PROGRAM PLC_PowerRF
VAR_INPUT
	nSocketType:UINT:=0;// socket 类型; 0 表示 server; 1 表示 client;
	sTerminalName:STRING;// 通讯对方名称 自定义
	sHost:STRING(20):='127.0.0.1';// 通讯IP地址; server时表示本地host; client时表示远程host
	nPort:UDINT:=8900;// 通讯端口号;
	bEnable:BOOL:=TRUE;// 通讯启用\禁用连接
	sSendSuffix:STRING:='';//此处可统一添加发送后缀字符 $R$N
	nQueueInterval:UDINT:=50;// 发送队列时间间隔 单位ms
	logHandleArray:ARRAY [1..5] OF POINTER TO printLogModule_EX;// log 操作 handle 数组
	logHandleArrayLength:UINT:=0;// log 操作 handle 数组长度, 不超过5
	readStateFlag:BOOL;
	ClearCom:BOOL;
	receiveFlag:BOOL;
END_VAR
VAR_OUTPUT
	bSendCondition	:BOOL;//可发送条件
	bSocketConnected:BOOL;//连接状态
END_VAR
VAR CONSTANT
	cNumBegin		:DINT:=1;
	cNumEnd			:DINT:=100;
END_VAR
VAR
	sendDataArray	:ARRAY [cNumBegin..cNumEnd] OF STRING(255);
	length			:DINT:=0;
	endPoint		:DINT:=cNumBegin;
	popupSendData	:STRING(255);
	//popup
	popupStep		:UINT:=0;
	popupTON1		:TON;
	popupTON2		:TON;
	iPopup			:DINT:=0;
	_PopupLength	:DINT:=0;
END_VAR
VAR
	tcpipClient					:tcpipClientModule_EX;
	tcpipServer					:tcpipServerModule_EX;////定义服务器对象
	
	tcpipSendDataBuff_Server	:STRING(255);//发送数据 Buff server
	tcpipSendDataBuff_Client	:STRING(255);//发送数据 Buff client
	
	tcpipSendDataClear			:STRING(255);//发送数据 清空
	tcpipSendData				:STRING(255);//发送数据
	
	tcpipRecDataBuff_Server		:STRING(255);//已接收数据 Buff server
	tcpipRecDataBuff_Client		:STRING(255);//已接收数据 Buff client
	
	tcpipRecDataClear			:STRING(255);//已接收数据 清空
	tcpipRecData				:STRING(255);//已接收数据
	
	tcpConnectR_Trig			:R_Trig;//初始连接上升沿
	tcpConnectF_Trig			:F_Trig;//初始连接下降沿
	registerStep				:UDINT;//ALC注册控制步
	registerTON					:TON;//ALC注册延时
	
	logHandleArray_index		:UINT:=1;
END_VAR
VAR
	bTrig_Start:BOOL;
	rTrig_Start:R_TRIG;
	tTrig_Start:TON;
	
	bTrig_Stop:BOOL;
	rTrig_Stop:R_TRIG;
	tTrig_Stop:TON;
	
	bTrig_Reset:BOOL;
	rTrig_Reset:R_TRIG;
	tTrig_Reset:TON;
	
	
	bTrig_Init:BOOL;
	rTrig_Init:R_TRIG;
	
	bTrig_All_Home:BOOL;
	rTrig_All_Home:R_TRIG;
	
	bTrig_Z_Safe:BOOL;
	rTrig_Z_Safe:R_TRIG;
	
	bTrig_P_Pos_:BOOL;
	rTrig_P_Pos_:R_TRIG;
	nTrig_P_Pos_TrayNum:UINT:=1;
	nTrig_P_Pos_RowNum:UINT:=1;
	
	bTrig_Move_P_:BOOL;
	rTrig_Move_P_:R_TRIG;
	nTrig_Move_P_TrayNum:UINT:=1;
	nTrig_Move_P_RowNum:UINT:=1;
	nTrig_Move_P_PosNum:UINT:=1;
	findposstart	:INT;
	findposend		:INT;
	find_pos		:INT;
	recStrTemp		:STRING(255);
END_VAR


CASE nSocketType OF
0://TCPIP server
	tcpipServer(
		sSrvNetId:= , 
		sLocalHost:=sHost , 
		nLocalPort:=nPort , 
		bStartConnect:=bEnable , 
		tcpipSDataLen:=TO_UDINT(LEN(tcpipSendDataBuff_Server)) , 
		tcpipSData:=ADR(tcpipSendDataBuff_Server) , 
		bSend:= , 
		tcpipRecDataLen:=SIZEOF(tcpipRecDataBuff_Server) , 
		tcpipRecData:=ADR(tcpipRecDataBuff_Server) , 
		bAccepted=> , 
		bSendBusy=> , 
		bRecData=> );
	bSendCondition:=tcpipServer.bAccepted AND NOT tcpipServer.bSendBusy;
	//TCPIP连接
	bSocketConnected:=tcpipServer.bAccepted;
	IF NOT tcpipServer.bAccepted THEN
		length:=0;
		endPoint:=cNumBegin;
	END_IF
	tcpConnectR_Trig(CLK:=tcpipServer.bAccepted);
	tcpConnectF_Trig(CLK:=tcpipServer.bAccepted);

1://TCPIP client
	tcpipClient(
		sSrvNetId:= , 
		sRemoteHost:=sHost , 
		nRemotePort:=nPort , 
		bStartConnect:=bEnable , 
		tcpipSDataLen:=TO_UDINT(LEN(tcpipSendDataBuff_Client)) , 
		tcpipSData:=ADR(tcpipSendDataBuff_Client) , 
		bSend:= , 
		tcpipRecDataLen:=SIZEOF(tcpipRecDataBuff_Client) , 
		tcpipRecData:=ADR(tcpipRecDataBuff_Client) , 
		bConnected=> , 
		bSendBusy=> , 
		bRecData=> );
	bSendCondition:=tcpipClient.bConnected AND NOT tcpipClient.bSendBusy;
	//TCPIP连接
	bSocketConnected:=tcpipClient.bConnected;
	IF NOT tcpipClient.bConnected THEN
		length:=0;
		endPoint:=cNumBegin;
	END_IF
	tcpConnectR_Trig(CLK:=tcpipClient.bConnected);
	tcpConnectF_Trig(CLK:=tcpipClient.bConnected);
END_CASE
IF ClearCom THEN
	length:=0;
	endPoint:=cNumBegin;
	ClearCom:=FALSE;
END_IF
IF tcpConnectR_Trig.Q THEN
	FOR logHandleArray_index:=1 TO logHandleArrayLength DO
		logHandleArray[logHandleArray_index]^.append(CONCAT(sTerminalName, ' has been connected'));
	END_FOR
	registerStep:=10;
END_IF
IF tcpConnectF_Trig.Q THEN
	FOR logHandleArray_index:=1 TO logHandleArrayLength DO
		logHandleArray[logHandleArray_index]^.append(CONCAT(sTerminalName, ' has been disconnected'));
	END_FOR
	registerStep:=0;
END_IF
//数据接收处理
CASE nSocketType OF
0://TCPIP server
	IF tcpipServer.bRecData THEN
		tcpipRecData:=tcpipRecDataBuff_Server;//buff转存
		tcpipRecDataBuff_Server:=tcpipRecDataClear;//转存之后清空buff
		dataProcessing();
	END_IF
1://TCPIP client
	IF tcpipClient.bRecData THEN
		tcpipRecData:=tcpipRecDataBuff_Client;//buff转存
		tcpipRecDataBuff_Client:=tcpipRecDataClear;//转存之后清空buff
		dataProcessing();
	END_IF
END_CASE


popup();

CASE registerStep OF
0:
	//Ready
END_CASE

METHOD appendSend : BOOL
VAR_INPUT
	str			:STRING(255);
END_VAR
VAR
	suffix					:STRING;
	strTemp_appendSend		:STRING(255);
END_VAR

IF endPoint>(cNumEnd-1) THEN
	RETURN;
END_IF
suffix:=sSendSuffix;//此处可统一添加发送后缀字符 $R$N

strTemp_appendSend:=CONCAT(str,suffix);
sendDataArray[endPoint]:=strTemp_appendSend;

endPoint:=endPoint+1;
length:=endPoint-cNumBegin;
END_METHOD

METHOD dataProcessing : BOOL
VAR_INPUT
END_VAR
VAR
	strTemp:STRING;
END_VAR
FOR logHandleArray_index:=1 TO logHandleArrayLength DO
	CASE nSocketType OF
	0://TCPIP server
//		logHandleArray[logHandleArray_index]^.append(CONCAT(CONCAT(CONCAT('Recevie From ', sTerminalName), ' -- '),tcpipRecData));
	1://TCPIP client
//		logHandleArray[logHandleArray_index]^.append(CONCAT(CONCAT(CONCAT('Recevie From ', sTerminalName), ' -- '),tcpipRecData));
	END_CASE
END_FOR
receiveFlag:=TRUE;
findposend:=0;
find_pos:=0;
IF MID(tcpipRecData,1,32)='$R' AND MID(tcpipRecData,1,33)='$R'  THEN
	gICP.PowerRF.controlMode:=STRING_TO_INT(MID(tcpipRecData,1,1));
	gICP.PowerRF.outputMode:=STRING_TO_INT(MID(tcpipRecData,1,2));
	gICP.PowerRF.outputState:=STRING_TO_INT(MID(tcpipRecData,1,3));
	strTemp:='';
	strTemp:=CONCAT(strTemp,(MID(tcpipRecData,2,6)));
	gICP.PowerRF.alarmState:=STRING_TO_INT(strTemp);
	strTemp:='';
	strTemp:=CONCAT(strTemp,(MID(tcpipRecData,5,9)));
	gICP.PowerRF.setpowerRead:=STRING_TO_UDINT(strTemp);
	strTemp:='';
	strTemp:=CONCAT(strTemp,(MID(tcpipRecData,5,15)));
	gICP.PowerRF.forwardpower:=STRING_TO_UDINT(strTemp);
	strTemp:='';
	strTemp:=CONCAT(strTemp,(MID(tcpipRecData,5,21)));
	gICP.PowerRF.reflectedpower:=STRING_TO_UDINT(strTemp);
	strTemp:='';
	strTemp:=CONCAT(strTemp,(MID(tcpipRecData,5,27)));
	gICP.PowerRF.maxpower:=STRING_TO_UDINT(strTemp);
	readStateFlag:=TRUE;
END_IF
END_METHOD

METHOD PRIVATE popup : BOOL
VAR_INPUT
END_VAR
CASE popupStep OF
0:
	IF length>0 AND bSendCondition THEN
		_PopupLength:=length;
		popupSendData:=sendDataArray[cNumBegin];
		FOR iPopup:=cNumBegin TO (_PopupLength-1) DO
			sendDataArray[iPopup]:=sendDataArray[iPopup+1];
		END_FOR
		endPoint:=endPoint-1;
		length:=endPoint-cNumBegin;
		sendData(popupSendData);//此处是调用信息发送
		popupStep:=10;
	END_IF
10:
	popupTON2(IN:=NOT popupTON2.Q, PT:=T#2S);
	IF NOT bSendCondition OR popupTON2.Q THEN
		popupTON2(IN:=FALSE);
		popupStep:=11;
	END_IF
11:
	IF bSendCondition THEN
		popupStep:=12;
	END_IF
	popupTON1(IN:=FALSE);
12:
	//popupTON1(IN:=NOT popupTON1.Q,PT:=T#10MS);
	popupTON1(IN:=NOT popupTON1.Q,PT:=TO_TIME(nQueueInterval));
	IF popupTON1.Q THEN
		popupStep:=0;
	END_IF
END_CASE
END_METHOD

METHOD ReadState : BOOL
VAR_INPUT
END_VAR
VAR
END_VAR
appendSend('Q$R');
END_METHOD

METHOD PRIVATE sendData : BOOL
VAR_INPUT
	dataStruct	:STRING(255);
END_VAR
IF bSendCondition AND bEnable THEN
	tcpipSendData:=dataStruct;
	
	CASE nSocketType OF
	0://TCPIP server
		tcpipSendDataBuff_Server:=tcpipSendData;
		tcpipSendData:=tcpipSendDataClear;	
		tcpipServer.bSend:=TRUE;
	1://TCPIP client
		tcpipSendDataBuff_Client:=tcpipSendData;
		tcpipSendData:=tcpipSendDataClear;	
		tcpipClient.bSend:=TRUE;
	END_CASE
	
	FOR logHandleArray_index:=1 TO logHandleArrayLength DO
		CASE nSocketType OF
		0://TCPIP server
//			logHandleArray[logHandleArray_index]^.append(CONCAT(CONCAT(CONCAT('Send To ', sTerminalName), ' -- '),tcpipSendDataBuff_Server));
		1://TCPIP client
//			logHandleArray[logHandleArray_index]^.append(CONCAT(CONCAT(CONCAT('Send To ', sTerminalName), ' -- '),tcpipSendDataBuff_Client));
		END_CASE
	END_FOR
END_IF
END_METHOD

METHOD WriteMaxPower : BOOL
VAR_INPUT
	maxpowerpoint:UDINT;
END_VAR
VAR
	str:STRING;
	_bit:UDINT;
	_ten:UDINT;
	_hundred:UDINT;
	_thousand:UDINT;
END_VAR
str:='';
_thousand:=maxpowerpoint/1000;
str:=CONCAT(str,UDINT_TO_STRING(maxpowerpoint));
//_hundred:=maxpowerpoint/100 MOD 10;
//str:=CONCAT(str,UDINT_TO_STRING(_hundred));
//_ten:=maxpowerpoint/10 MOD 10;
//str:=CONCAT(str,UDINT_TO_STRING(_ten));
//_bit:=maxpowerpoint MOD 10;
//str:=CONCAT(str,UDINT_TO_STRING(_bit));
str:=CONCAT(str,' M$R');
appendSend(str);
END_METHOD

METHOD WritePower : BOOL
VAR_INPUT
	powerpoint:UDINT;
END_VAR
VAR
	str:STRING;
	_bit:UDINT;
	_ten:UDINT;
	_hundred:UDINT;
	_thousand:UDINT;
END_VAR
str:='';
//_thousand:=powerpoint/1000;
str:=CONCAT(str,UDINT_TO_STRING(powerpoint));
//_hundred:=powerpoint/100 MOD 10;
//str:=CONCAT(str,UDINT_TO_STRING(_hundred));
//_ten:=powerpoint/10 MOD 10;
//str:=CONCAT(str,UDINT_TO_STRING(_ten));
//_bit:=powerpoint MOD 10;
//str:=CONCAT(str,UDINT_TO_STRING(_bit));
str:=CONCAT(str,' W$R');
appendSend(str);
END_METHOD

METHOD WriteReset : BOOL
VAR_INPUT
		

END_VAR
appendSend('RESET$R');
END_METHOD

METHOD WriteRS232Mode : BOOL
VAR_INPUT
		

END_VAR
appendSend('***$R');
END_METHOD

METHOD WriteStart : BOOL
VAR_INPUT
		

END_VAR
appendSend('G$R');
END_METHOD

METHOD WriteStop : BOOL
VAR_INPUT
		

END_VAR
appendSend('S$R');
END_METHOD

END_PROGRAM

(* stored: Version 1.1.0.1, ProductVersion 3.1.4024.4
   POU PLC_PowerRF: Id {85380df0-8fdb-48e1-aff9-ca76d02218cf}, SpecialFunc None
   Folder CMD: Id {8b38d363-c970-4008-9462-e4673db2cac3}
   Folder Recevie: Id {7910003a-7a4e-46a1-9b57-3f00a440373b}
   Folder Send: Id {348e8ae3-9132-4cfe-8e14-5fedb96fdd51}
   Folder Private: Id {e004de8c-6536-4ed7-a070-f75304a20453}
   Method appendSend: Id {f3074b24-86b6-487e-a04b-90021562abe2}
   Method dataProcessing: Id {a4ea7910-cee5-4312-8b32-651085150e25}
   Method popup: Id {6ee42d8a-ab2c-444d-87df-63743ac19fea}
   Method ReadState: Id {5a0e8dd1-df0f-4f1e-980e-f0ec72be7cc7}
   Method sendData: Id {715bc88a-50de-4cdc-a499-bdf58dd8d340}
   Method WriteMaxPower: Id {f8e0f3de-cfc1-4a18-aa91-6390688bcad9}
   Method WritePower: Id {8e939e86-cd63-4e56-9bc8-935c9c8958c6}
   Method WriteReset: Id {69dd7ba4-2596-4024-90ec-3e4651863b34}
   Method WriteRS232Mode: Id {80e0a6ba-a3a2-46a9-b186-da1bb90a8dac}
   Method WriteStart: Id {360cd40d-a4c2-484a-bd75-c13f5c8a28dd}
   Method WriteStop: Id {ad465910-4516-4624-9d2a-ed27213fc374} *)
